// Mitsubishi GX Works2 project: 0708-비교연산   PLC: Q02/Q02H

PROGRAM MAIN
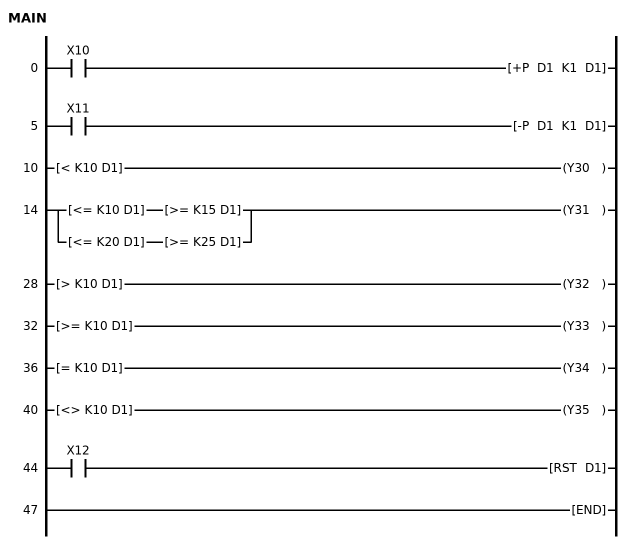
0     LD      X10
      +P      D1 K1 D1
5     LD      X11
      -P      D1 K1 D1
10    LD<     K10 D1
      OUT     Y30
14    LD<=    K10 D1
      AND>=   K15 D1
      LD<=    K20 D1
      AND>=   K25 D1
      ORB
      OUT     Y31
28    LD>     K10 D1
      OUT     Y32
32    LD>=    K10 D1
      OUT     Y33
36    LD=     K10 D1
      OUT     Y34
40    LD<>    K10 D1
      OUT     Y35
44    LD      X12
      RST     D1
47    END
END_PROGRAM
